{attribute 'pack_mode' := '1'}
TYPE
  ST_OpcUa_LrealPoint EXTENDS ST_OpcUa_PointBase :
  STRUCT
    Value : LREAL;
  END_STRUCT
END_TYPE

(* stored: Version 1.1.0.1, ProductVersion 3.1.4024.9
   DUT ST_OpcUa_LrealPoint: Id {a5014129-d7e3-4112-8513-2048ff39cac2} *)
